{attribute addProperty BoxType "EL3443-0000-0016"}
{attribute addProperty Id "Active_PowerAT %I*REAL32417Apparent_PowerAT %I*REAL32418Reactive_PowerAT %I*REAL32419Power_FactorAT %I*REAL32420"}
{attribute addProperty CRC "3905309348"}
{attribute addProperty SizeInBites "128"}
{attribute addProperty SizeInBytes "16"}
TYPE L1_Power_E8C64AA4 :
STRUCT
	{attribute addProperty Name "Active_Power"}
	Active_Power AT %I* : REAL;
	{attribute addProperty Name "Apparent_Power"}
	Apparent_Power AT %I* : REAL;
	{attribute addProperty Name "Reactive_Power"}
	Reactive_Power AT %I* : REAL;
	{attribute addProperty Name "Power_Factor"}
	Power_Factor AT %I* : REAL;
END_STRUCT
END_TYPE

(* stored: Version 1.2.0.0, ProductVersion 3.1.4024.9
   DUT L1_Power_E8C64AA4: Id {21c624dd-bdd8-41aa-8efc-b7ce221990ee} *)
